// Mitsubishi GX Works2 project: COMPLETE(1)   PLC: Q02/Q02H

// task Task_01 (event TRUE, interval 0, priority 31): POU_01

PROGRAM POU_01
VAR
  MAIN : POINTER;
END_VAR
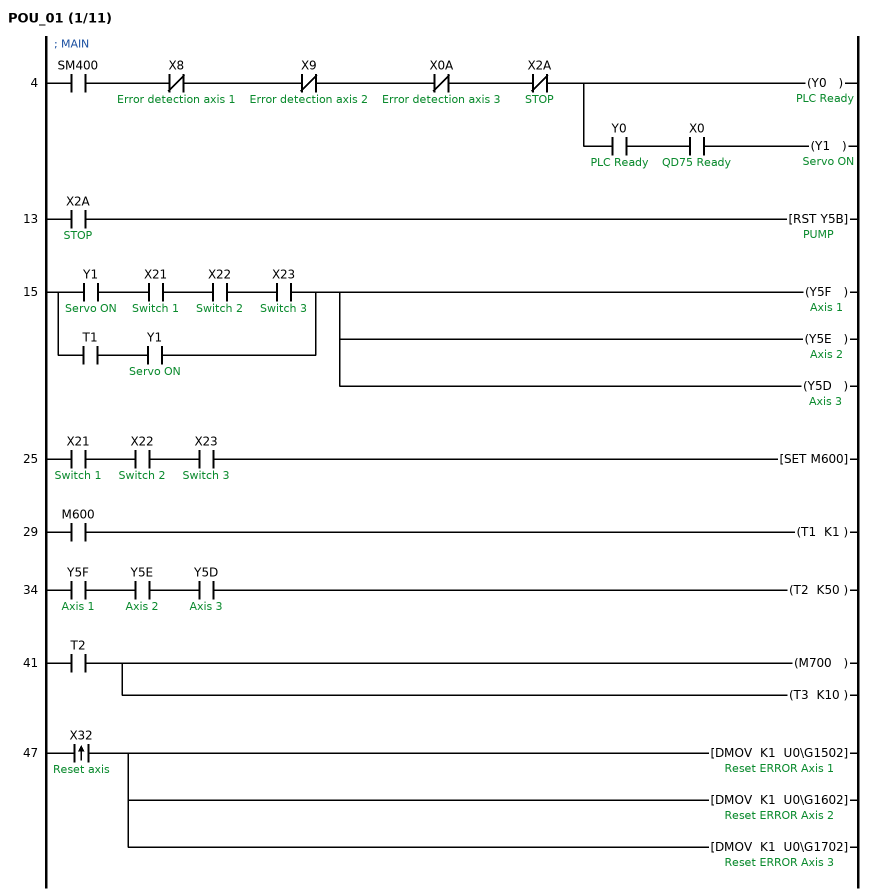
; MAIN
4     LD      SM400
      ANI     X8  ; Error detection axis 1
      ANI     X9  ; Error detection axis 2
      ANI     X0A  ; Error detection axis 3
      ANI     X2A  ; STOP
      OUT     Y0  ; PLC Ready
      AND     Y0  ; PLC Ready
      AND     X0  ; QD75 Ready
      OUT     Y1  ; Servo ON
13    LD      X2A  ; STOP
      RST     Y5B  ; PUMP
15    LD      Y1  ; Servo ON
      AND     X21  ; Switch 1
      AND     X22  ; Switch 2
      AND     X23  ; Switch 3
      LD      T1
      AND     Y1  ; Servo ON
      ORB
      OUT     Y5F  ; Axis 1
      OUT     Y5E  ; Axis 2
      OUT     Y5D  ; Axis 3
25    LD      X21  ; Switch 1
      AND     X22  ; Switch 2
      AND     X23  ; Switch 3
      SET     M600
29    LD      M600
      OUT     T1 K1
34    LD      Y5F  ; Axis 1
      AND     Y5E  ; Axis 2
      AND     Y5D  ; Axis 3
      OUT     T2 K50
41    LD      T2
      OUT     M700
      OUT     T3 K10
47    LDP     X32  ; Reset axis
      DMOV    K1 U0\G1502  ; Reset ERROR Axis 1
      DMOV    K1 U0\G1602  ; Reset ERROR Axis 2
      DMOV    K1 U0\G1702  ; Reset ERROR Axis 3
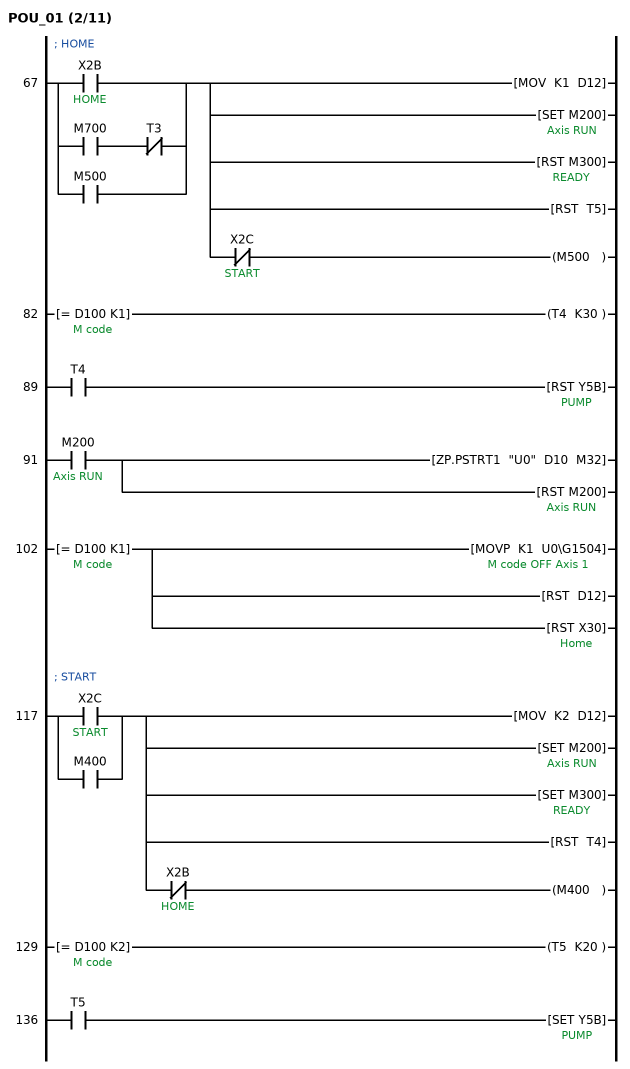
; HOME
67    LD      X2B  ; HOME
      LD      M700
      ANI     T3
      ORB
      OR      M500
      MOV     K1 D12
      SET     M200  ; Axis RUN
      RST     M300  ; READY
      RST     T5
      ANI     X2C  ; START
      OUT     M500
82    LD=     D100 K1  ; M code
      OUT     T4 K30
89    LD      T4
      RST     Y5B  ; PUMP
91    LD      M200  ; Axis RUN
      ZP.PSTRT1 "U0" D10 M32
      RST     M200  ; Axis RUN
102   LD=     D100 K1  ; M code
      MOVP    K1 U0\G1504  ; M code OFF Axis 1
      RST     D12
      RST     X30  ; Home
; START
117   LD      X2C  ; START
      OR      M400
      MOV     K2 D12
      SET     M200  ; Axis RUN
      SET     M300  ; READY
      RST     T4
      ANI     X2B  ; HOME
      OUT     M400
129   LD=     D100 K2  ; M code
      OUT     T5 K20
136   LD      T5
      SET     Y5B  ; PUMP
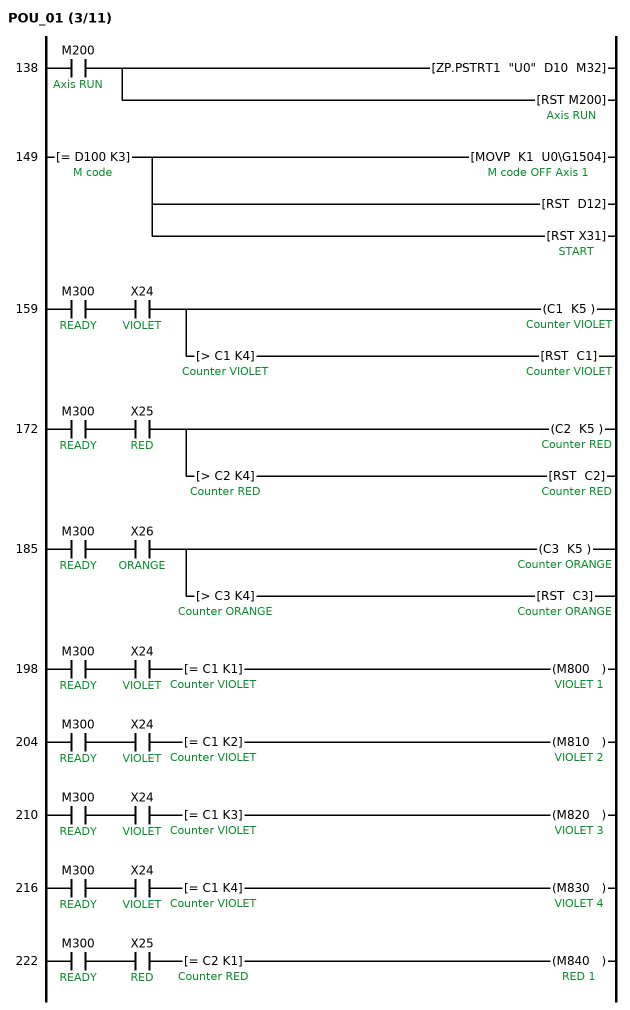
138   LD      M200  ; Axis RUN
      ZP.PSTRT1 "U0" D10 M32
      RST     M200  ; Axis RUN
149   LD=     D100 K3  ; M code
      MOVP    K1 U0\G1504
      RST     D12
      RST     X31  ; START
159   LD      M300  ; READY
      AND     X24  ; VIOLET
      OUT     C1 K5  ; Counter VIOLET
      AND>    C1 K4  ; Counter VIOLET
      RST     C1  ; Counter VIOLET
172   LD      M300  ; READY
      AND     X25  ; RED
      OUT     C2 K5  ; Counter RED
      AND>    C2 K4  ; Counter RED
      RST     C2  ; Counter RED
185   LD      M300  ; READY
      AND     X26  ; ORANGE
      OUT     C3 K5  ; Counter ORANGE
      AND>    C3 K4  ; Counter ORANGE
      RST     C3  ; Counter ORANGE
198   LD      M300  ; READY
      AND     X24  ; VIOLET
      AND=    C1 K1  ; Counter VIOLET
      OUT     M800  ; VIOLET 1
204   LD      M300  ; READY
      AND     X24  ; VIOLET
      AND=    C1 K2  ; Counter VIOLET
      OUT     M810  ; VIOLET 2
210   LD      M300  ; READY
      AND     X24  ; VIOLET
      AND=    C1 K3  ; Counter VIOLET
      OUT     M820  ; VIOLET 3
216   LD      M300  ; READY
      AND     X24  ; VIOLET
      AND=    C1 K4  ; Counter VIOLET
      OUT     M830  ; VIOLET 4
222   LD      M300  ; READY
      AND     X25  ; RED
      AND=    C2 K1  ; Counter RED
      OUT     M840  ; RED 1
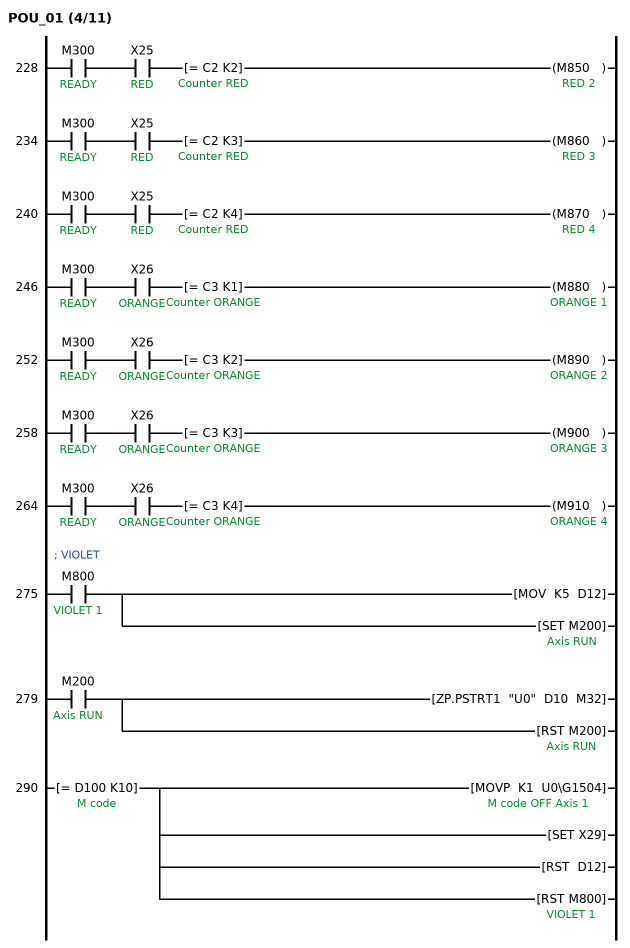
228   LD      M300  ; READY
      AND     X25  ; RED
      AND=    C2 K2  ; Counter RED
      OUT     M850  ; RED 2
234   LD      M300  ; READY
      AND     X25  ; RED
      AND=    C2 K3  ; Counter RED
      OUT     M860  ; RED 3
240   LD      M300  ; READY
      AND     X25  ; RED
      AND=    C2 K4  ; Counter RED
      OUT     M870  ; RED 4
246   LD      M300  ; READY
      AND     X26  ; ORANGE
      AND=    C3 K1  ; Counter ORANGE
      OUT     M880  ; ORANGE 1
252   LD      M300  ; READY
      AND     X26  ; ORANGE
      AND=    C3 K2  ; Counter ORANGE
      OUT     M890  ; ORANGE 2
258   LD      M300  ; READY
      AND     X26  ; ORANGE
      AND=    C3 K3  ; Counter ORANGE
      OUT     M900  ; ORANGE 3
264   LD      M300  ; READY
      AND     X26  ; ORANGE
      AND=    C3 K4  ; Counter ORANGE
      OUT     M910  ; ORANGE 4
; VIOLET
275   LD      M800  ; VIOLET 1
      MOV     K5 D12
      SET     M200  ; Axis RUN
279   LD      M200  ; Axis RUN
      ZP.PSTRT1 "U0" D10 M32
      RST     M200  ; Axis RUN
290   LD=     D100 K10  ; M code
      MOVP    K1 U0\G1504
      SET     X29
      RST     D12
      RST     M800  ; VIOLET 1
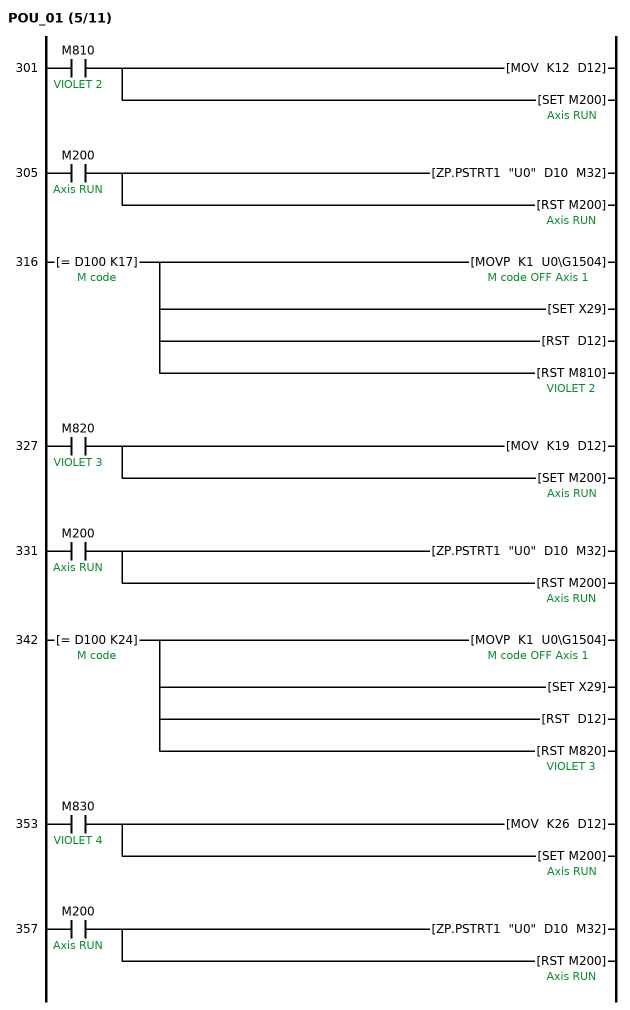
301   LD      M810  ; VIOLET 2
      MOV     K12 D12
      SET     M200  ; Axis RUN
305   LD      M200  ; Axis RUN
      ZP.PSTRT1 "U0" D10 M32
      RST     M200  ; Axis RUN
316   LD=     D100 K17  ; M code
      MOVP    K1 U0\G1504
      SET     X29
      RST     D12
      RST     M810  ; VIOLET 2
327   LD      M820  ; VIOLET 3
      MOV     K19 D12
      SET     M200  ; Axis RUN
331   LD      M200  ; Axis RUN
      ZP.PSTRT1 "U0" D10 M32
      RST     M200  ; Axis RUN
342   LD=     D100 K24  ; M code
      MOVP    K1 U0\G1504
      SET     X29
      RST     D12
      RST     M820  ; VIOLET 3
353   LD      M830  ; VIOLET 4
      MOV     K26 D12
      SET     M200  ; Axis RUN
357   LD      M200  ; Axis RUN
      ZP.PSTRT1 "U0" D10 M32
      RST     M200  ; Axis RUN
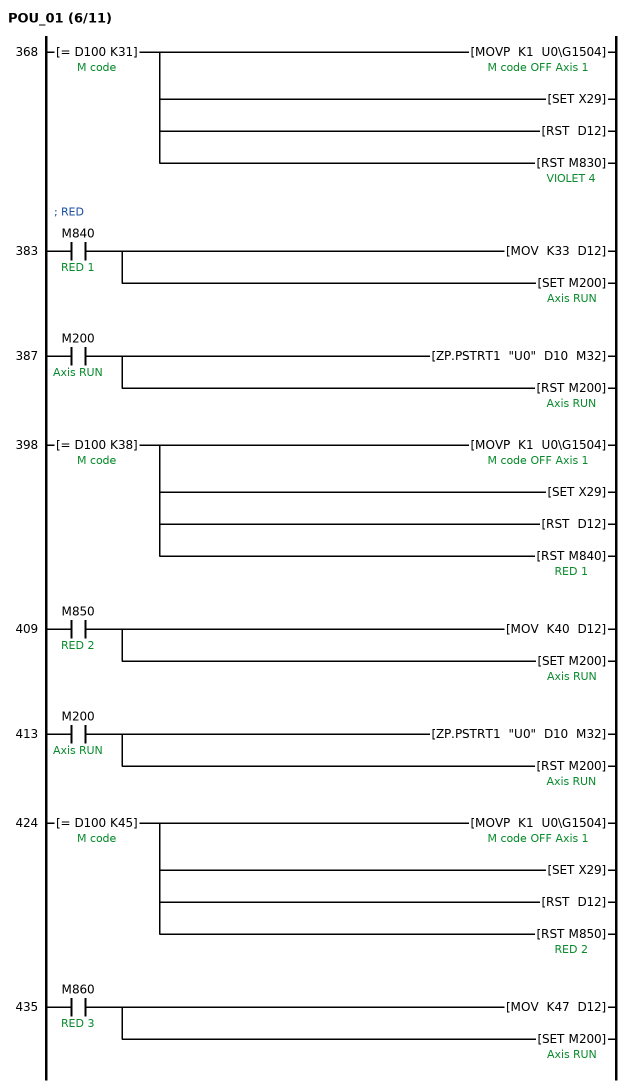
368   LD=     D100 K31  ; M code
      MOVP    K1 U0\G1504
      SET     X29
      RST     D12
      RST     M830  ; VIOLET 4
; RED
383   LD      M840  ; RED 1
      MOV     K33 D12
      SET     M200  ; Axis RUN
387   LD      M200  ; Axis RUN
      ZP.PSTRT1 "U0" D10 M32
      RST     M200  ; Axis RUN
398   LD=     D100 K38  ; M code
      MOVP    K1 U0\G1504
      SET     X29
      RST     D12
      RST     M840  ; RED 1
409   LD      M850  ; RED 2
      MOV     K40 D12
      SET     M200  ; Axis RUN
413   LD      M200  ; Axis RUN
      ZP.PSTRT1 "U0" D10 M32
      RST     M200  ; Axis RUN
424   LD=     D100 K45  ; M code
      MOVP    K1 U0\G1504
      SET     X29
      RST     D12
      RST     M850  ; RED 2
435   LD      M860  ; RED 3
      MOV     K47 D12
      SET     M200  ; Axis RUN
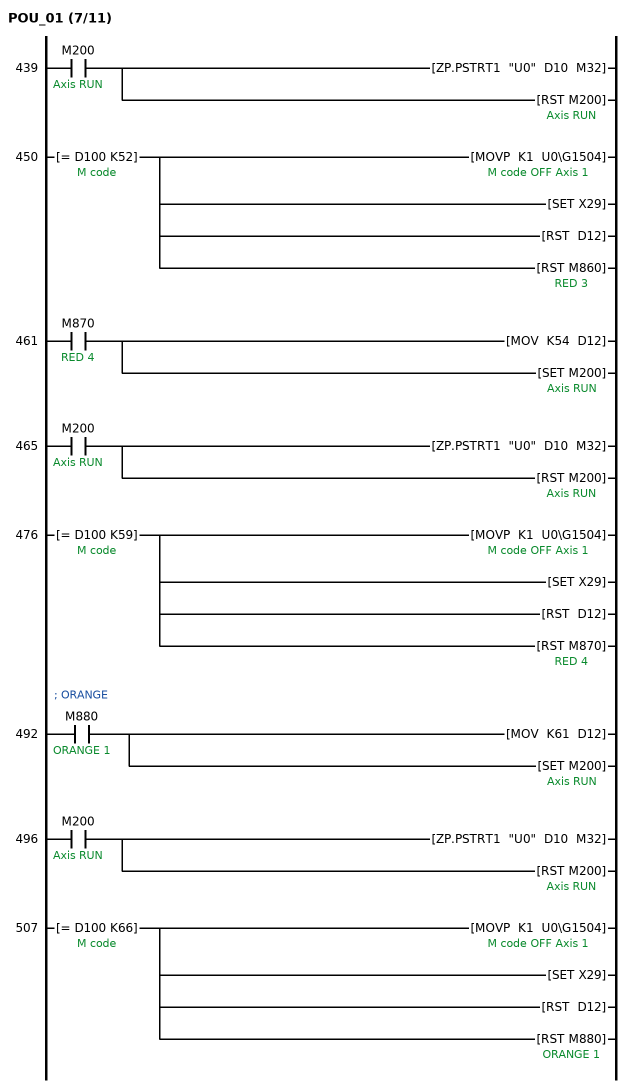
439   LD      M200  ; Axis RUN
      ZP.PSTRT1 "U0" D10 M32
      RST     M200  ; Axis RUN
450   LD=     D100 K52  ; M code
      MOVP    K1 U0\G1504
      SET     X29
      RST     D12
      RST     M860  ; RED 3
461   LD      M870  ; RED 4
      MOV     K54 D12
      SET     M200  ; Axis RUN
465   LD      M200  ; Axis RUN
      ZP.PSTRT1 "U0" D10 M32
      RST     M200  ; Axis RUN
476   LD=     D100 K59  ; M code
      MOVP    K1 U0\G1504
      SET     X29
      RST     D12
      RST     M870  ; RED 4
; ORANGE
492   LD      M880  ; ORANGE 1
      MOV     K61 D12
      SET     M200  ; Axis RUN
496   LD      M200  ; Axis RUN
      ZP.PSTRT1 "U0" D10 M32
      RST     M200  ; Axis RUN
507   LD=     D100 K66  ; M code
      MOVP    K1 U0\G1504
      SET     X29
      RST     D12
      RST     M880  ; ORANGE 1
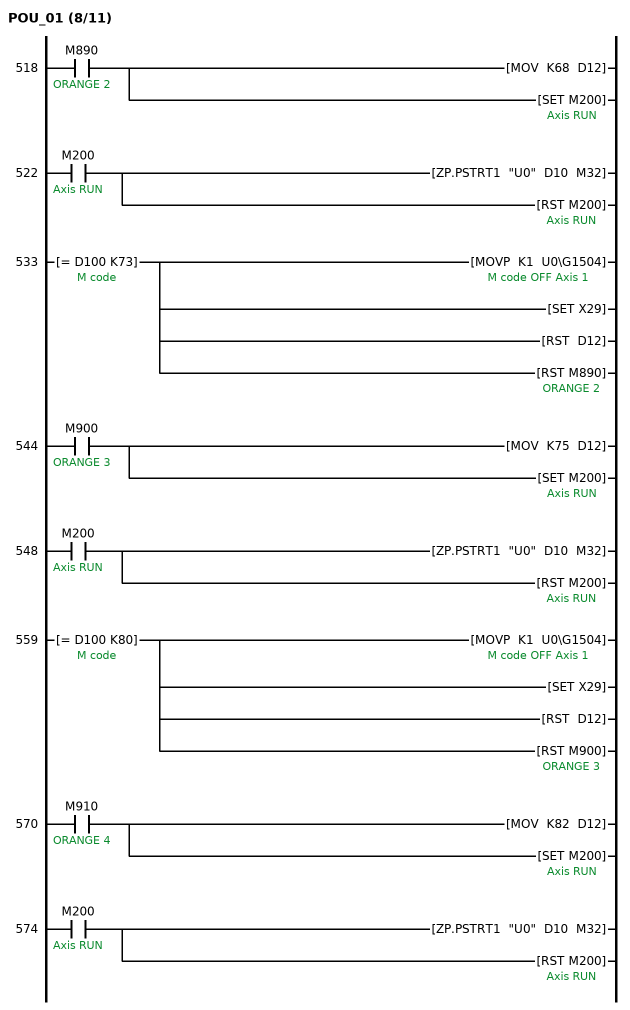
518   LD      M890  ; ORANGE 2
      MOV     K68 D12
      SET     M200  ; Axis RUN
522   LD      M200  ; Axis RUN
      ZP.PSTRT1 "U0" D10 M32
      RST     M200  ; Axis RUN
533   LD=     D100 K73  ; M code
      MOVP    K1 U0\G1504
      SET     X29
      RST     D12
      RST     M890  ; ORANGE 2
544   LD      M900  ; ORANGE 3
      MOV     K75 D12
      SET     M200  ; Axis RUN
548   LD      M200  ; Axis RUN
      ZP.PSTRT1 "U0" D10 M32
      RST     M200  ; Axis RUN
559   LD=     D100 K80  ; M code
      MOVP    K1 U0\G1504
      SET     X29
      RST     D12
      RST     M900  ; ORANGE 3
570   LD      M910  ; ORANGE 4
      MOV     K82 D12
      SET     M200  ; Axis RUN
574   LD      M200  ; Axis RUN
      ZP.PSTRT1 "U0" D10 M32
      RST     M200  ; Axis RUN
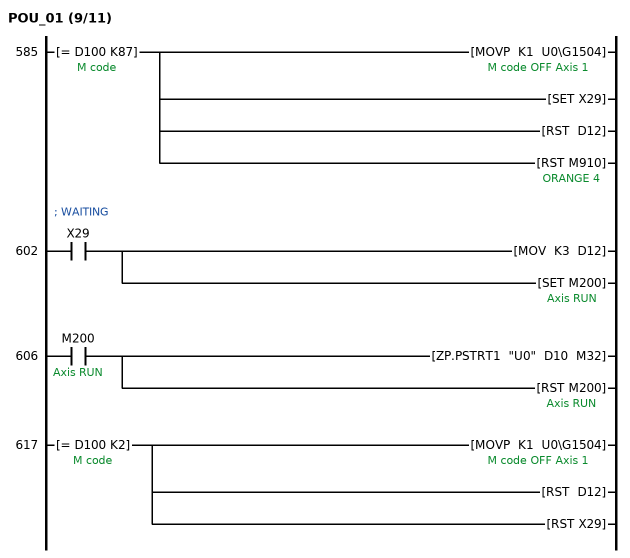
585   LD=     D100 K87  ; M code
      MOVP    K1 U0\G1504
      SET     X29
      RST     D12
      RST     M910  ; ORANGE 4
; WAITING
602   LD      X29
      MOV     K3 D12
      SET     M200  ; Axis RUN
606   LD      M200  ; Axis RUN
      ZP.PSTRT1 "U0" D10 M32
      RST     M200  ; Axis RUN
617   LD=     D100 K2  ; M code
      MOVP    K1 U0\G1504
      RST     D12
      RST     X29
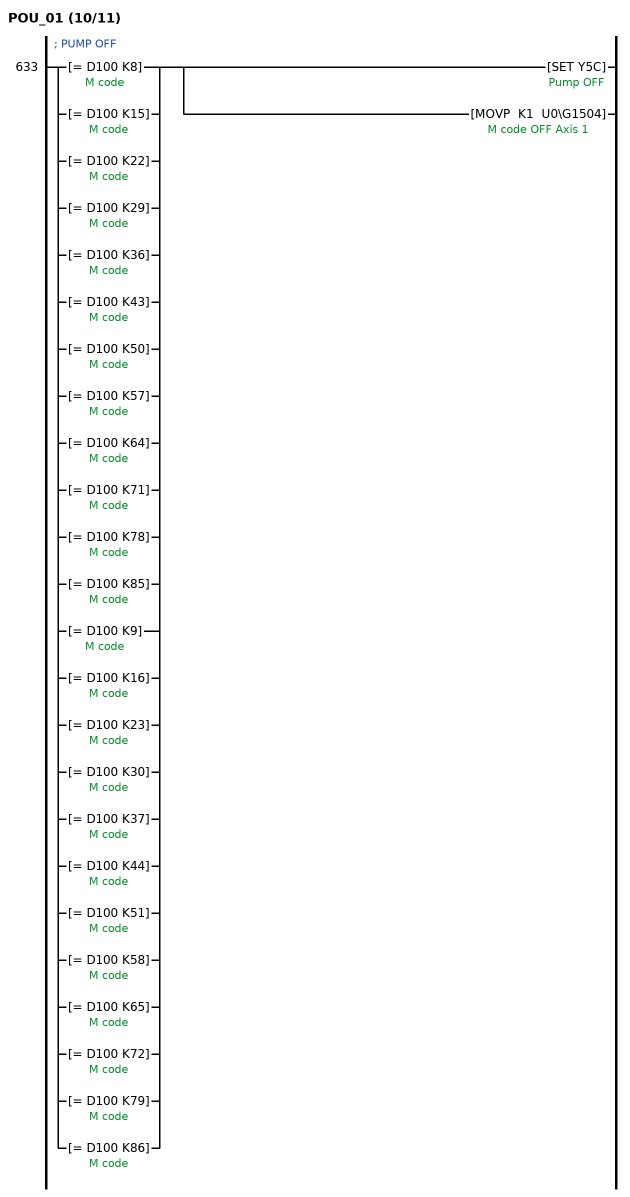
; PUMP OFF
633   LD=     D100 K8  ; M code
      OR=     D100 K15  ; M code
      OR=     D100 K22  ; M code
      OR=     D100 K29  ; M code
      OR=     D100 K36  ; M code
      OR=     D100 K43  ; M code
      OR=     D100 K50  ; M code
      OR=     D100 K57  ; M code
      OR=     D100 K64  ; M code
      OR=     D100 K71  ; M code
      OR=     D100 K78  ; M code
      OR=     D100 K85  ; M code
      OR=     D100 K9  ; M code
      OR=     D100 K16  ; M code
      OR=     D100 K23  ; M code
      OR=     D100 K30  ; M code
      OR=     D100 K37  ; M code
      OR=     D100 K44  ; M code
      OR=     D100 K51  ; M code
      OR=     D100 K58  ; M code
      OR=     D100 K65  ; M code
      OR=     D100 K72  ; M code
      OR=     D100 K79  ; M code
      OR=     D100 K86  ; M code
      SET     Y5C  ; Pump OFF
      MOVP    K1 U0\G1504
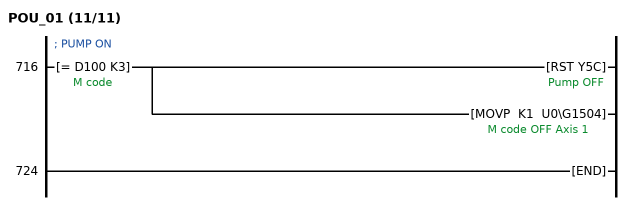
; PUMP ON
716   LD=     D100 K3  ; M code
      RST     Y5C  ; Pump OFF
      MOVP    K1 U0\G1504
724   END
END_PROGRAM

// device comments not shown above
X5  ; JOG Axis 1
X6  ; JOG Axis 2
X7  ; JOG Axis 3
X1F  ; Servo ON
X28  ; Sensor NPN
X33  ; Start DC
X40  ; YELLOW 4
M10  ; Reset ERROR Axis
M15  ; Home
M16  ; Homing
Y50  ; DC
Y51  ; RASP
D200  ; Counter RED
D300  ; Counter ORANGE
D400  ; Counter VIOLET
